{attribute 'qualified_only'}
VAR_GLOBAL
	ThermalCouple	: ARRAY[1..12] OF ST_ThermalCouple;
	ChargerSP		: REAL;
	ChargerSP_norm	: REAL;
	ChargerSP_raw	: INT;
END_VAR

VAR_GLOBAL PERSISTENT
	TemperatureSP 					: REAL;
	TemperatureSP_norm				: REAL;
	TemperatureSP_raw				: REAL;
	
END_VAR

(* stored: Version 1.1.0.1, ProductVersion 3.1.4024.11
   GVL MCP_IO: Id {2eccccd0-d6b2-453f-b49b-33f7d0364904} *)
